// Mitsubishi GX Works2 project: 機電整合乙級第四題-ST   PLC: FX3U/FX3UC

// task Task_01 (event TRUE, interval 0, priority 31): POU_01

PROGRAM POU_01
VAR
  wProgramStep : INT;
  wSpeed : INT;
  wXPulse : INT;
  wYPulse : INT;
  bL1Full : BOOL;
  bL2Full : BOOL;
  wInColor : INT;
  tdT143 : TON;
  tdT144 : TON;
  bM143 : BOOL;
  bM17 : BOOL;
  tdT23 : TON;
  bM0 : BOOL;
  arCellPos : ARRAY [0..3,0..1] OF INT;
  wInCount : INT;
  tdT21 : TON;
  tdT25 : TON;
  arCellColor : ARRAY [0..3] OF INT;
  arCellCount : ARRAY [0..3] OF INT;
  tdT24 : TON;
  tdT22 : TON;
  bM133 : BOOL;
END_VAR
(* 機電整合乙級術科第四題
   Author: Steven Luo
   Date: 2018/10/25
*)

IF M8000 THEN
	wSpeed := D1 * 1000;
END_IF;

IF M8002 THEN
	D1 := 3;
	(* X, Y postion in pulse *)
	arCellPos[0, 0] := 7800;  (* B->X *)
	arCellPos[0, 1] := 4400;  (* B->Y *)
	arCellPos[1, 0] := 14850; (* A->X *)
	arCellPos[1, 1] := 4400;  (* A->Y *)
	arCellPos[2, 0] := 14850; (* C->X *)
	arCellPos[2, 1] := 12300; (* C->Y *)
	arCellPos[3, 0] := 7800;  (* D->X *)
	arCellPos[3, 1] := 12300; (* D->Y *)
	wXPulse := 15440;
	wYPulse := 4098;
	bM143 := FALSE;
	wProgramStep := 0;
END_IF;

IF M133 THEN
	bM133 := TRUE;
END_IF;

IF NOT M144 THEN
	IF bM0 THEN
		D5 := 0;
	ELSE
		D5 := 410;
	END_IF;
END_IF;

IF NOT X17 THEN (* 急停 *)
	ZRST(TRUE, Y4, Y17);
	ZRST(TRUE, D0, D50);
	ZRST(TRUE, M20 ,M23);
	M8349 := TRUE;
	M8359 := TRUE;
	D5 := 413;
	bM17 := TRUE;
	M144 := FALSE;
	wProgramStep := -1;
END_IF;

IF X17 AND bM17 THEN (* 解除急停，按下復歸 *)
	D5 := 412;
	IF M132 THEN
		M8349 := FALSE;
		M8359 := FALSE;
		bM17 := FALSE;
		bM143 := TRUE;
		tdT143(IN := FALSE);
		tdT144(IN := FALSE);
		wProgramStep := 100;
	END_IF;
END_IF;

IF bM143 THEN (* 黃燈閃爍 *)
	tdT143(IN := NOT tdT144.Q, PT := T#500ms);
	tdT144(IN := tdT143.Q, PT := T#500ms);
	M143 := tdT143.Q;
END_IF;

OUT(X10 AND X4 AND X5 AND X6, bM0); (* 原點條件 *)

OUT(bL1Full, M145);
OUT(bL2Full, M146);

PLSR(M20, wSpeed, wXPulse, 300, Y0);
OUT(M22, Y2);
PLSR(M21, wSpeed, wYPulse, 300, Y1);
OUT(M23, Y3);

CASE wProgramStep OF
0:
	IF X17 THEN
		IF M130 THEN
			wProgramStep := 200;
		ELSE
			wProgramStep := 20;
		END_IF;
	END_IF;
20:
	IF M130 THEN
		wProgramStep := 0;
	END_IF;
	IF bM0 THEN
		D0 := 0;
		D5 := 0;
		ZRST(TRUE, D10, D13);
		ZRST(TRUE, M151, M165);
		FOR D20 := 0 TO 3 BY 1 DO
			arCellColor[D20] := 0;
			arCellCount[D20] := 0;
		END_FOR;
		bM133 := FALSE;
		M1 := FALSE;
		M142 := TRUE;
		M144 := FALSE;
		bL1Full := FALSE;
		bL2Full := FALSE;
		wInColor := 0;
		wInCount := 0;
		tdT21(IN := FALSE);
		tdT22(IN := FALSE);
		tdT23(IN := FALSE);
		tdT24(IN := FALSE);
		tdT25(IN := FALSE);
		IF M131 THEN
			IF NOT X0 THEN
				D5 := 411;
			END_IF;
			M1 := TRUE;
			M142 := FALSE;
			M144 := TRUE;
			wProgramStep := 21;
		END_IF;
	END_IF;
21:
	IF bM133 THEN
		wProgramStep := 0;
		RETURN;
	END_IF;
	IF X0 THEN (* 有料 *)
		ZRST(TRUE, M147, M149);
		Y4 := TRUE; (* 進料缸進料 *)
		tdT21(IN := TRUE, PT := T#2s);
		IF tdT21.Q THEN
			Y4 := FALSE;
			IF X1 OR X2 OR X3 THEN
				D0 := D0 + 1;
				IF X1 THEN
					M147 := TRUE;
					wInColor := 1;
				ELSIF X2 THEN
					M148 := TRUE;
					wInColor := 2;
				ELSIF X3 THEN
					M149 := TRUE;
					wInColor := 3;
				END_IF;
				wProgramStep := 22;
			ELSE
				wProgramStep := 0;
			END_IF;
		END_IF;
	END_IF;
22:
	IF WORD_TO_INT(D0) > 4 THEN
		FOR D20 := 0 TO 3 BY 1 DO
			IF (arCellColor[D20] = wInColor) AND (arCellCount[D20] = 1) THEN
				EXIT;
			END_IF;
		END_FOR;
		IF D20 > 3 THEN
			tdT22(IN := TRUE, PT := T#2s);
			IF tdT22.Q THEN
				tdT21(IN := FALSE);
				tdT22(IN := FALSE);
				wProgramStep := 21;
			END_IF;
			RETURN;
		END_IF;
	END_IF;
	Y5 := TRUE; (* Z軸氣壓缸下降 *)
	IF X7 THEN (* Z軸中位 *)
		wProgramStep := 23;
	END_IF;
23:
	tdT23(IN := TRUE, PT := T#500ms);
	IF tdT23.Q THEN
		Y6 := TRUE; (* 氣壓夾爪夾 *)
		wProgramStep := 24;
	END_IF;
24:
	tdT24(IN := TRUE, PT := T#500ms);
	IF tdT24.Q THEN
		Y5 := FALSE; (* Z軸氣壓缸上升 *)
		IF X6 THEN
			IF WORD_TO_INT(D0) <= 4 THEN
				wXPulse := arCellPos[wInCount, 0];
				wYPulse := arCellPos[wInCount, 1];
			ELSE
				wXPulse := arCellPos[D20, 0];
				wYPulse := arCellPos[D20, 1];
			END_IF;
			OUT(TRUE, M20);
			OUT(TRUE, M21);
			OUT(TRUE, M23);
			D5 := 410;
			wProgramStep := 25;
		END_IF;
	END_IF;
25:
	tdT25(IN := TRUE, PT := T#2s);
	IF tdT25.Q THEN
		IF NOT M8340 AND NOT M8350 THEN
			M20 := FALSE;
			M21 := FALSE;
			M23 := FALSE;
			wProgramStep := 26;
		END_IF;
	END_IF;
26:
	Y5 := TRUE; (* Z軸氣壓缸下降 *)
	IF X7 THEN (* Z軸中位 *)
		Y6 := FALSE;
		Y7 := TRUE; (* 氣壓夾爪放 *)
		IF WORD_TO_INT(D0) <= 4 THEN
			arCellColor[wInCount] := wInColor;
			arCellCount[wInCount] := 1;
			CASE wInCount OF
			0:
				D11 := D11 + 1;
				CASE wInColor OF
				1:
					M155 := TRUE;
				2:
					M156 := TRUE;
				3:
					M157 := TRUE;
				END_CASE;
			1:
				D10 := D10 + 1;
				CASE wInColor OF
				1:
					M151 := TRUE;
				2:
					M152 := TRUE;
				3:
					M153 := TRUE;
				END_CASE;
			2:
				D12 := D12 + 1;
				CASE wInColor OF
				1:
					M159 := TRUE;
				2:
					M160 := TRUE;
				3:
					M161 := TRUE;
				END_CASE;
			3:
				D13 := D13 + 1;
				CASE wInColor OF
				1:
					M163 := TRUE;
				2:
					M164 := TRUE;
				3:
					M165 := TRUE;
				END_CASE;
			END_CASE;
		ELSE
			arCellCount[D20] := arCellCount[D20] + 1;
			CASE D20 OF
			0:
				D11 := D11 + 1;
			1:
				D10 := D10 + 1;
			2:
				D12 := D12 + 1;
			3:
				D13 := D13 + 1;
			END_CASE;
		END_IF;
		wProgramStep := 27;
	END_IF;
27:
	Y5 := FALSE; (* Z軸氣壓缸上升 *)
	IF X6 THEN
		Y7 := FALSE;
		wInCount := wInCount + 1;
		IF wInCount = 4 THEN
			IF D0 = 4 THEN
				bL1Full := TRUE;
			ELSIF WORD_TO_INT(D0) >= 8 THEN
				bL2Full := TRUE;
			END_IF;
			wInCount := 0;
		END_IF;
		wXPulse := 32000;
		wYPulse := 32000;
		wProgramStep := 201; (* 回原點 *)
	END_IF;
100:
	IF M132 THEN
		D1 := 3;
		wXPulse := 32000;
		wYPulse := 32000;
		wProgramStep := 201; (* 自動復歸 *)
	END_IF;
200:
	wXPulse := 32000;
	wYPulse := 32000;
	OUT(M110, Y4);
	IF X6 THEN
		OUT(M111 OR M112, M20);
		OUT(M112 AND NOT M111, M22);
		OUT(M113 OR M114, M21);
		OUT(M113 AND NOT M114, M23);
	END_IF;
	RST(M115, Y5);
	SET(M116, Y5);
	OUT(M117, Y6);
	OUT(M118, Y7);
	IF NOT M130 THEN
		wProgramStep := 0;
	END_IF;
201:
	OUT(NOT X4, M20);
	OUT(NOT X4, M22);
	IF X4 THEN
		D8140 := 0;
	END_IF;
	OUT(NOT X5, M21);
	IF X5 THEN
		D8142 := 0;
	END_IF;
	IF bM0 THEN
		D5 := 0;
		IF bM143 THEN
			bM143 := FALSE;
			M143 := FALSE;
			wProgramStep := 0;
		ELSE
			IF M1 THEN
				tdT21(IN := FALSE);
				tdT23(IN := FALSE);
				tdT24(IN := FALSE);
				tdT25(IN := FALSE);
				wProgramStep := 21;
			ELSE
				wSpeed := D1 * 1000;
				wProgramStep := 200;
			END_IF;
		END_IF;
	END_IF;
END_CASE;
END_PROGRAM
